TEXTLIST textListBottom
  0 = ''
  1 = 'X'
  2 = 'Λ'
  3 = 'V'
   = ''
END_TEXTLIST

(* stored: Version 1.1.0.1, ProductVersion 3.1.4024.11
   TextList textListBottom: Id {11be4c82-d48b-0a38-0775-fb047d04c765} *)
